// TIA Portal V20 export
TYPE "typeEnMeterValues"
TITLE = Energy Meter Werte / Energy meter value
// Struktur Energy Meter Werte / Structure energy meter values
// stored: Access Published
   STRUCT
      dataRecordVersion : Byte;   // dataRecordVersion
      reserved : Byte;   // Reserve / Reserved
      voltageL1N : Real;   // Spannung L1N / Voltage L1N
      voltageL2N : Real;   // Spannung L2N / Voltage L2N
      voltageL3N : Real;   // Spannung L3N / Voltage L3N
      voltageL1L2 : Real;   // Spannung L1L2 / Voltage L1L2
      voltageL2L3 : Real;   // Spannung L2L3 / Voltage L2L3
      voltageL3L1 : Real;   // Spannung L3L1 / Voltage L3L1
      currentL1 : Real;   // Strom L1 / Current L1
      currentL2 : Real;   // Strom L2 / Current L2
      currentL3 : Real;   // Strom L3 / Current L3
      powerFactorL1 : Real;   // Leistunsfaktor L1 / Power factor L1
      powerFactorL2 : Real;   // Leistunsfaktor L2 / Power factor L2
      powerFactorL3 : Real;   // Leistunsfaktor L3 / Power factor L3
      powerFactorOverall : Real;   // Leistunsfaktor Gesamt / Power factor Overall
      frequency : Real;   // Frequenz / Frequency
      voltageSymmetry : Real;   // Spannungs-Symetrie / Voltage symmetry
      currentSymmetry : Real;   // Strom-Symetrie / Current symmetry
      apparentPowerL1 : Real;   // Scheinleistung L1 / Apparent power L1
      apparentPowerL2 : Real;   // Scheinleistung L2 / Apparent power L2
      apparentPowerL3 : Real;   // Scheinleistung L3 / Apparent power L3
      apparentPowerOverall : Real;   // Scheinleistung Gesamt / Apparent power Overall
      reactivePowerL1 : Real;   // Blindleistung L1 / Reactive power L1
      reactivePowerL2 : Real;   // Blindleistung L2 / Reactive power L2
      reactivePowerL3 : Real;   // Blindleistung L3 / Reactive power L3
      reactivePowerOverall : Real;   // Blindleistung Geamt / Reactive power Overall
      effectivePowerL1 : Real;   // Wirkleistung L1 / Effective power L1
      effectivePowerL2 : Real;   // Wirkleistung L2 / Effective power L2
      effectivePowerL3 : Real;   // Wirkleistung L3 / Effective power L3
      effectivePowerOverall : Real;   // Wirkleistung Gesamz / Effective power Overall
      phaseAngleL1 : Real;   // Phasen Winkel L1 / Phase angle L1
      phaseAngleL2 : Real;   // Phasen Winkel L2 / Phase angle L2
      phaseAngleL3 : Real;   // Phasen Winkel L3 / Phase angle L3
      appEnOverall32bit : Real;   // Energie Scheinleistung Gesamt 32bit / Apparent energy overall 32bit
      reaEnOverall32bit : Real;   // Energie Blindleistung Gesamt 32bit / Reactive energy overall 32bit
      effEnOverall32bit : Real;   // Energie Wirkleistung Gesamt 32bit / Effective energy overall 32bit
      reaEnImport32bit : Real;   // Energie Blindleistung Import 32bit / Reactive energy import 32bit
      reaEnExport32bit : Real;   // Energie Blindleistung Export 32bit / Reactive energy export 32bit
      effEnImport32bit : Real;   // Energie Wirkleistung Import 32bit / Effective energy import 32bit
      effEnExport32bit : Real;   // Energie Wirkleistung Export 32bit / Effective energy export 32bit
      appEnOverall64bit : LReal;   // Energie Scheinleistung Gesamt 64bit / Apparent energy overall 64bit
      reaEnOverall64bit : LReal;   // Energie Blindleistung Gesamt 64bit / Reactive energy overall 64bit
      effEnOverall64bit : LReal;   // Energie Wirkleistung Gesamt 64bit / Effective energy overall 64bit
      reaEnImport64bit : LReal;   // Energie Blindleistung Import 64bit / Reactive energy import 64bit
      reaEnExport64bit : LReal;   // Energie Blindleistung Export 64bit / Reactive energy export 64bit
      effEnImport64bit : LReal;   // Energie Wirkleistung Import 64bit / Effective energy import 64bit
      effEnExport64bit : LReal;   // Energie Wirkleistung Export 64bit / Effective energy export 64bit
   END_STRUCT;
END_TYPE
